FUNCTION_BLOCK FB_Safety_module
VAR_INPUT
END_VAR
VAR_OUTPUT
END_VAR
VAR
	SI_0	: UINT;
	SI_1	: UINT;
	GI_0 	: UINT;
	GI_1 	: UINT;
	safety_status	: SafetyStatus	:= SafetyStatus.UNKNOWN;
	
	station_mode	: StationMode;
	iStationMode	: UINT;
	iState: INT;
	bEstop_detection	: BOOL;	
	
	ton_timeout	: TON;	
	eStates					:	E_SafetyStates	:=	E_SafetyStates.IDLE;
	iStateTemp			: INT;
	errorMessage	: STRING;
	xError	: BOOL;
	eStates_safetyDoor	: E_SAFETYDOOR	:= E_SAFETYDOOR.IDLE;
	
	
	
	
	
	GPWM	: FB_GPWM;
	GPWM_1s	: FB_GPWM;
	tonSaftyDelay: TON;
	b_EStopRestarting  : BOOL;
	T_EStopRestart : TON;
//////////////////////SAFETY hardware config///////////////	
	mcp_estop	: BOOL;
	mcp_safetyDoor	: BOOL;
	belt_estop	: BOOL;
	lift_estop : BOOL;
	lift_lightCurtain_left	: BOOL;
	lift_lightCurtain_right	: BOOL;
	lift_station_detection	: BOOL;
	
	robot_EES				: BOOL;
	robot_EAS				: BOOL;
	buffer_safety			: BOOL;
	loading_safety			: BOOL;
	working_safety			: BOOL;
//	buffer_safety_24v		: BOOL;
//	buffer_safety_stepmotor	: BOOL;
//	loding_safety_sto		: BOOL;
//	loding_safety_24v		: BOOL;
//	working_safety_sto		: BOOL;
//	working_safety_24v		: BOOL;
	
	ref_safety_door	: POINTER TO ST_safetyDoor;
	safety_door_unlock_en		: BOOL;
END_VAR

M_mapping();
M_safetyDoor();
xError	:=NOT(robot_EES AND buffer_safety AND loading_safety AND working_safety); //if only open the door,machine will just stop,so can control the machine munually
//to do:as below commit and reprogram safety project and test

CASE iState	 OF
	0:
	;

	2:
		IF update_station_mode(2) THEN
			iState	:= 0;
		END_IF	
	3:
		IF M_reset() THEN
			iState	:= 0;
		END_IF
		
END_CASE
//安全Safety报警 确认 复位
tonSaftyDelay(IN:= NOT tonSaftyDelay.Q ,PT:=T#1S);
b_ErrorAck := tonSaftyDelay.Q;



GPWM(i_xEnable:=TRUE,i_udiTime:=25,i_udiCycle:=50);
GPWM_1s(i_xEnable:=TRUE,i_udiTime:=500,i_udiCycle:=1000);
//light curtain mute
GVL.fb_working.lightcurtain_mute_left 	:= GVL.fb_buffer.fb_rollers[3].sensor_mute.Q OR GVL.fb_loading.roller_x.photo_sensor_mute_left.Q;   
GVL.fb_working.lightcurtain_mute_right 	:= GVL.fb_loading.roller_x.photo_sensor_mute_right.Q OR GVL.fb_working.roller_inbound.photo_sensor_mute.Q;
 


 //EDM config
 SPtop_EDM  	  	   := TRUE ;  
 robot_eas_edm  	   := TRUE ;
 light_STO_EDM         := TRUE ;
 PickModule_STO_EDM    := TRUE ;
 Rolller_belt_STO_EDM  := TRUE ;

PROPERTY _stationMode : StationMode
GET
_stationMode	:= station_mode;
END_GET
SET
station_mode	:= _stationMode;
END_SET
END_PROPERTY

METHOD M_mapping : BOOL
VAR_INPUT
END_VAR



mcp_estop					:= SI0_0 AND SI0_1;
mcp_safetyDoor				:= SI0_2 AND SI0_3;
belt_estop					:= SI1_0 AND SI1_1;
lift_lightCurtain_left		:= SI2_0 AND SI2_1;
lift_estop					:= SI2_2 AND SI2_3;
lift_lightCurtain_right		:= SI3_0 AND SI3_1;
lift_station_detection		:= SI3_2 AND SI3_3;
bShield_light_curtain_Left	:= SI4_0;
bShield_light_curtain_Right	:= SI4_1;


robot_EES				:= SO0_0;
robot_EAS				:= SO0_1;
buffer_safety			:= SO1_0;

loading_safety			:= SO2_0;

working_safety			:= SO3_0;

	
	                    
                    
                  
	
IF robot_EES AND robot_EAS THEN 
    safety_status := SafetyStatus.READY ;   //正常
ELSE
	safety_status := SafetyStatus.SAFETY_STOPPED; //急停状态
END_IF

GI_0.0	:= GVL.fb_mcp.st_safety_door.button_reset;
GI_0.1	:= GVL.fb_mcp.st_safety_door.button_unlock;
GI_0.2	:= GVL.fb_mcp.st_safety_door.door_closed;

SI_0.0	:= mcp_estop;
SI_0.1	:= mcp_safetyDoor;
SI_0.2	:= belt_estop;
SI_0.3	:= lift_estop;
SI_0.4	:= lift_station_detection;
END_METHOD

METHOD M_reset : BOOL
VAR_INPUT
	
END_VAR
M_reset	:= FALSE;
//check if all estop
//check if safety door ossd
//check if safety door closed
//lock safety door 
//reset to output safety
//////////////////////////////////////////////////////////timeout//////////////////////////////////////////
ton_timeout();
IF eStates<>E_SafetyStates.IDLE AND eStates<>E_SafetyStates.ERROR  THEN
	IF iStateTemp=eStates THEN
		ton_timeout.IN	:=TRUE;
	ELSE
		ton_timeout.IN	:=FALSE;
		iStateTemp	:= eStates;
	END_IF
ELSE
	ton_timeout.IN	:=FALSE;
END_IF
IF ton_timeout.Q THEN	
	ton_timeout.IN	:=FALSE;
	CASE eStates OF
		E_SafetyStates.DOOR_LOCK:		
			errorMessage	:= CONCAT('door lock error.->safety ',INT_TO_STRING(iStateTemp));
	END_CASE
	IF eStates=E_SafetyStates.DOOR_LOCK AND eStates<>E_SafetyStates.TRIG_RESET THEN
		eStates	:= E_SafetyStates.ERROR;
	END_IF
	
END_IF
CASE eStates OF
	E_SafetyStates.IDLE:
		xError	:= FALSE;
		eStates	:= E_SafetyStates.CHECK_ESTOP;
	E_SafetyStates.CHECK_ESTOP:
		IF mcp_estop AND belt_estop AND lift_estop THEN
			eStates	:= E_SafetyStates.CHECK_DOOR_CLOSED;
		ELSE
			eStates	:= E_SafetyStates.ERROR;
		END_IF
	E_SafetyStates.CHECK_DOOR_CLOSED:
		IF GVL.fb_mcp.st_safety_door.door_closed THEN
			eStates	:= E_SafetyStates.DOOR_LOCK;
		ELSE
			eStates	:= E_SafetyStates.ERROR;
		END_IF
	E_SafetyStates.DOOR_LOCK:
		ref_safety_door^.door_lock	:= FALSE;
		IF mcp_safetyDoor THEN
			eStates	:= E_SafetyStates.TRIG_RESET;
		END_IF		
	E_SafetyStates.TRIG_RESET:
		ton_timeout.PT	:= T#2S;
		b_EStopRestart	:= GPWM.q_xOut;
		IF ton_timeout.Q THEN
			b_EStopRestart	:= FALSE;
			eStates	:= E_SafetyStates.CHECK_SAFETY_OUTPUT;
		END_IF
	E_SafetyStates.CHECK_SAFETY_OUTPUT:	
		IF robot_EES AND robot_EAS AND buffer_safety AND loading_safety AND working_safety THEN
			eStates	:= E_SafetyStates.DONE;
		ELSE
			eStates	:= E_SafetyStates.ERROR;
		END_IF
	E_SafetyStates.DONE:
		M_reset	:= TRUE;
		eStates	:= E_SafetyStates.IDLE;
	E_SafetyStates.ERROR:	
		M_reset	:= TRUE;
		xError	:= TRUE;
		eStates	:= E_SafetyStates.IDLE;

	
END_CASE
END_METHOD

METHOD M_safetyDoor : BOOL
VAR_INPUT
END_VAR
ref_safety_door	:= ADR(GVL.fb_mcp.st_safety_door);
safety_door_unlock_en	:= safety_status=SafetyStatus.SAFETY_STOPPED OR station_mode = StationMode.STOPPED OR station_mode = StationMode.DISABLED
							OR station_mode = StationMode.FORCE_STOP OR station_mode = StationMode.INTERVENTION;

							
CASE eStates_safetyDoor	 OF
	E_SAFETYDOOR.IDLE:
		IF mcp_safetyDoor THEN
			eStates_safetyDoor	:= E_SAFETYDOOR.LOCKED;
		ELSE
			eStates_safetyDoor	:= E_SAFETYDOOR.UNLOCKED;
		END_IF
	E_SAFETYDOOR.LOCKED:
		ref_safety_door^.lamp_reset	:=	FALSE;
		ref_safety_door^.lamp_unlock	:= FALSE;
		IF ref_safety_door^.button_unlock THEN
			eStates_safetyDoor	:= E_SAFETYDOOR.UNLOCKING;
		END_IF
	E_SAFETYDOOR.REQUEST_LOCK:
	;
	E_SAFETYDOOR.SAFETY:
	;
	E_SAFETYDOOR.UNLOCKED:
		ref_safety_door^.lamp_unlock	:= TRUE;//door unlocked,unlock lamp solid
		IF ref_safety_door^.door_closed THEN
			ref_safety_door^.lamp_reset	:= GPWM_1s.q_xOut;//door closed,reset lamp blinking
			IF ref_safety_door^.button_reset THEN
				eStates_safetyDoor	:= E_SAFETYDOOR.WAIT_LOCKED;
			END_IF
		ELSE
			ref_safety_door^.lamp_reset	:= FALSE;
		END_IF
	E_SAFETYDOOR.WAIT_LOCKED:
		ref_safety_door^.door_lock	:= FALSE;
		IF mcp_safetyDoor THEN
			eStates_safetyDoor	:= E_SAFETYDOOR.LOCKED;
	 	END_IF
	E_SAFETYDOOR.UNLOCKING:
		ref_safety_door^.lamp_unlock	:= GPWM_1s.q_xOut;//door opennig,unlock lamp blinking
		IF safety_door_unlock_en THEN
			ref_safety_door^.door_lock	:= TRUE;
			IF NOT mcp_safetyDoor THEN
				eStates_safetyDoor	:= E_SAFETYDOOR.UNLOCKED;
			END_IF
		END_IF
	
END_CASE
END_METHOD

{attribute 'TcRpcEnable'}
METHOD update_station_mode  : BOOL
VAR_INPUT
	iMode	: StationMode;
END_VAR
update_station_mode	:= FALSE;
station_mode	:= iMode;
update_station_mode	:= TRUE;
END_METHOD

END_FUNCTION_BLOCK

(* stored: Version 1.1.0.1, ProductVersion 3.1.4024.12
   POU FB_Safety_module: Id {589679bc-3a60-44ea-a3dd-41af04fbe7bf}, SpecialFunc None
   Property _stationMode: Id {fa1a69a3-64f3-40be-8c11-e2e8d858f937}
   Get Get: Id {d232f638-792a-4a6e-932a-82e7dde798a5}
   Set Set: Id {2d1fc079-c675-4ec2-9cbe-a441bd46a266}
   Method M_mapping: Id {d65f4aa6-b391-4ff2-83f9-f1479fd3c9f4}
   Method M_reset: Id {8b41f1d7-fa71-4d85-b5b2-adf9e9a2f81c}
   Method M_safetyDoor: Id {9ae49d5b-b993-491d-87e3-565117d40da3}
   Method update_station_mode: Id {64d128c5-2a5a-4d16-9d84-da9d84099763} *)
